FUNCTION_BLOCK FB_HardwareFFOutput
VAR
END_VAR

END_FUNCTION_BLOCK

(* stored: Version 1.1.0.1, ProductVersion 3.1.4022.12
   POU FB_HardwareFFOutput: Id {8c2f0148-9967-4c03-964c-9a83e44c0f77}, SpecialFunc None *)
